FUNCTION_BLOCK FB_Component_HMI EXTENDS FB_BaseComponent_HMI IMPLEMENTS ITF_Component_HMI
VAR
	itfComponentConnector				: ITF_Component_HMI_Connector;
	refstComponentData					: reference to ST_Component_HMI;
END_VAR

END_FUNCTION_BLOCK

(* stored: Version 1.1.0.1, ProductVersion 3.1.4024.15
   POU FB_Component_HMI: Id {262cdf04-054e-404a-a25f-05e09b93d66c}, SpecialFunc None *)
